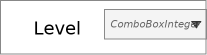
VISUALIZATION V_LevelSelecCmb  // 207x55
    ComboBoxInteger (104,9 103x30), variable: VisuGVL.fbPanelImp.Level, text list: 'LevelCmbTxtList'
    Label (5,2 105x53), "Level"
END_VISUALIZATION

(* stored: Version 1.1.0.1, ProductVersion 3.1.4024.4
   Visu V_LevelSelecCmb: Id {43974eb8-897b-432e-9a93-1e195d8db0ea} *)
